Universal Robots PolyScope program: move.urp

Program move (installation=default directory=/home/ur/ursim-current/programs createdIn=3.15.6.106324 lastSavedIn=3.15.6.106324 robotSerialNumber=2018339999)
Calibrated DH parameters: a=[0, -0.24365, -0.21325, 0, 0, 0]; d=[0.1519, 0, 0, 0.11235, 0.08535, 0.0819]; alpha=[1.570796, 0, 0, 1.570796, -1.570796, 0]; deltaTheta=[0, 0, 0, 0, 0, 0]
BeforeStart
  Set ExpressionOutput pin=register0; expression=0
Robot Program (runOnlyOnce=false)
  MoveJ speed 60 deg/s, acceleration 80 deg/s^2 (useActiveTCP=true)
    Waypoint Waypoint_1: TCP in base x=-118.696 y=-298.509 z=192.299 mm, rx=-0.0012 ry=3.1163 rz=0.0389 rad; joints [-91.592, -99.335, -113.614, -58.521, 91.396, -1.655] deg
  Set ExpressionOutput pin=register0; expression=101
  Set DigitalOutput pin=digital_out[0]; digitalValue=0
  MoveJ speed 60 deg/s, acceleration 80 deg/s^2 (useActiveTCP=true)
    Waypoint Waypoint_2: TCP in base x=45.634 y=-332.069 z=297.098 mm, rx=-0.1593 ry=3.1135 rz=0.0408 rad; joints [-63.072, -94.663, -89.257, -86.897, 91.855, 21.056] deg
  Set ExpressionOutput pin=register0; expression=202
  Set DigitalOutput pin=digital_out[0]; digitalValue=1
